(*
SPDX-FileCopyrightText: © 2026 Oleksandr Tiutyk <trofimich@gmail.com>
SPDX-License-Identifier: MIT
License: https://opensource.org/license/mit
*)

(*!
<summary>Static test adapter exposing the inherited formatter with deterministic inputs.</summary>
*)

FUNCTION_BLOCK ExceptionTimestampProbe EXTENDS TOF_Core.StandardException

METHOD FormatTimestamp : TOF_Core.ERROR_MESSAGE
VAR_INPUT
	mode : TOF_Core.TIMESTAMP_DISPLAY_MODE;
	localTime : LDATE_AND_TIME;
	utcTime : LDATE_AND_TIME;
END_VAR
AppendTimestampDescription(
	targetMessage := FormatTimestamp,
	timestampDisplayMode := mode,
	localTimestamp := localTime,
	utcTimestamp := utcTime
);
END_METHOD

END_FUNCTION_BLOCK

(* stored: Version 1.1.0.1
   POU ExceptionTimestampProbe: Id {eeec5711-a86f-436b-b43b-050f8522b132}, SpecialFunc None
   Method FormatTimestamp: Id {e6c4f6eb-9a61-4bbc-bc62-687bec77c8fb} *)
